FUNCTION_BLOCK FB_MoveVelocity_Test EXTENDS TcUnit.FB_TestSuite

TestCaseMove('Set Init',0, 0, 1000, 1000, TRUE);

TestCaseMove('Set Valid Motion_1',0, 1000, 1000, 1000, FALSE);
TestCaseMove('Set Valid Motion_2',0, 100, 1000, 1000, FALSE);
TestCaseMove('Set Valid Motion_3',0, 10, 1000, 1000, TRUE);	
TestCaseMove('Set Valid Motion_4',0, -1000, -1000, -1000, FALSE);
TestCaseMove('Set Valid Motion_5',0, -100, -1000, -1000, FALSE);
TestCaseMove('Set Valid Motion_6',0, -10, -1000, -1000, TRUE);

TestCaseMove('Set 2Zone Motion_1',-5, 1000, 1000, 1000, FALSE);
TestCaseMove('Set 2Zone Motion_2',-5, 100, 1000, 1000, FALSE);
TestCaseMove('Set 2Zone Motion_3',-5, 10, 2000, 2000, TRUE);	
TestCaseMove('Set 2Zone Motion_4',5, -1000, -1000, -1000, FALSE);
TestCaseMove('Set 2Zone Motion_5',5, -100, -1000, -1000, FALSE);
TestCaseMove('Set 2Zone Motion_6',5, -10, -2000, -2000, TRUE);

TestCaseMove('Set Dirty Motion_1',0, 10, 0.001, 0.001, FALSE);
TestCaseMove('Set Dirty Motion_2',0, 10, 0, 0, FALSE);
TestCaseMove('Set Dirty Motion_3',0, 10, 1E+12, 1E+12, TRUE);	
TestCaseMove('Set Dirty Motion_4',0, -1E+3, 1E+12, 1E+12, TRUE);	

TestCaseMove('Set Dirty ACC/DEC_1',0, 1000, -1000, -1000, FALSE);
TestCaseMove('Set Dirty ACC/DEC_2',0, 100, -1000, -1000, FALSE);
TestCaseMove('Set Dirty ACC/DEC_3',0, 10, -1000, -1000, TRUE);
TestCaseMove('Set Dirty ACC/DEC_4',0, -1000, 1000, 1000, FALSE);
TestCaseMove('Set Dirty ACC/DEC_5',0, -100, 1000, 1000, FALSE);
TestCaseMove('Set Dirty ACC/DEC_6',0, -10, 1000, 1000, TRUE);

METHOD TestCaseMove
VAR_INPUT
	sName 				: T_MaxString;
	fInitVelocity 		: REAL;
	fVelocity 			: REAL;
	fAcceleration 		: REAL;
	fDeceleration 		: REAL;
	bExpected 			: BOOL;
END_VAR

VAR
	fbMoveVelocity 		: FB_MoveVelocity;
	nCycleCount 		: INT;
	bResult 			: BOOL;
	fResult 			: REAL;
	fAcc 				: REAL;
	fExpectedAcc 		: REAL := 0;
END_VAR
TEST(sName);
	
fbMoveVelocity.fVelocity := fInitVelocity;

FOR nCycleCount := 0 TO 10 DO
    fbMoveVelocity(fTargetVelocity := fVelocity, fAccMax := fAcceleration, fDecMax := fDeceleration);
END_FOR;

bResult := fbMoveVelocity.bIsReached;
fResult := fbMoveVelocity.fVelocity;
fAcc := fbMoveVelocity.fAcc;

AssertEquals(Expected := bExpected,
             Actual := bResult,
             Message := 'Value is not reached');	
			 
IF bExpected THEN
	AssertEquals(Expected := fVelocity,
             Actual := fResult,
             Message := 'Velocity value is not correct');	
	AssertEquals(Expected := fExpectedAcc,
             Actual := fAcc,
             Message := 'Acc value is not correct');	
END_IF
	 
TEST_FINISHED();
END_METHOD

END_FUNCTION_BLOCK

(* stored: Version 1.1.0.1, ProductVersion 3.1.4024.12
   POU FB_MoveVelocity_Test: Id {22044dc0-8dc7-05bd-3f30-832d4a4177fd}, SpecialFunc None
   Method TestCaseMove: Id {45e9bff8-3120-05a7-27c5-ce7653ced786} *)
